// TIA Portal V19 export
DATA_BLOCK "ALARM DB"   // DB20
{ S7_Optimized_Access := 'FALSE' }
   VAR
      "EMERGENCY STOP" : Bool;
      "AIR FAIL" : Bool;
      "MGF FEED PUMP P-101 A MCB TRIP" : Bool;
      "MGF FEED PUMP P-101 B MCB TRIP" : Bool;
      "MGF BACK WASH  P-102 A MCB TRIP" : Bool;
      "MGF BACK WASH P-102 B MCB TRIP" : Bool;
      "UF FEED PUMP P-103 A MCB TRIP" : Bool;
      "UF FEED PUMP P-103 B MCB TRIP" : Bool;
      "UF BLOWER AB-201 A MCB TRIP" : Bool;
      "UF BLOWER AB-201 B MCB TRIP" : Bool;
      "DM FEED PUMP P-502 A MPCB TRIP" : Bool;
      "DM FEED PUMP P-502 B MPCB TRIP" : Bool;
      "DM FEED PUMP P-502 C MPCB TRIP" : Bool;
      "CIP P-601" : Bool;
      "BACK WASH RECOVERY P-801 A MPCB TRIP" : Bool;
      "BACK WASH RECOVERY P-801 B MPCB TRIP" : Bool;
      "UF BACKWASH P-201A TRIP" : Bool;
      "UF BACKWASH P-201B TRIP" : Bool;
      "MGF FEED PUMP P-101 A MCB_FEEDBACK FAIL" : Bool;
      "MGF FEED PUMP P-101 B MCB_FEEDBACK FAIL" : Bool;
      "MGF BACK WASH  P-102 A MCB_FEEDBACK FAIL" : Bool;
      "MGF BACK WASH P-102 B MCB_FEEDBACK FAIL" : Bool;
      "UF FEED PUMP P-103 A MCB_FEEDBACK FAIL" : Bool;
      "UF FEED PUMP P-103 B MCB_FEEDBACK FAIL" : Bool;
      "UF BLOWER AB-201 A MCB_FEEDBACK FAIL" : Bool;
      "UF BLOWER AB-201 B MCB_FEEDBACK FAIL" : Bool;
      "DM FEED PUMP P-502 A MPCB_FEEDBACK FAIL" : Bool;
      "DM FEED PUMP P-502 B MPCB_FEEDBACK FAIL" : Bool;
      "DM FEED PUMP P-502 C MPCB_FEEDBACK FAIL" : Bool;
      "CIP P-601_FEEDBACK FAIL" : Bool;
      "BACK WASH RECOVERY P-801 A MPCB_FEEDBACK FAIL" : Bool;
      "BACK WASH RECOVERY P-801 B MPCB_FEEDBACK FAIL" : Bool;
      "UF BACKWASH P-201A_FEEDBACK FAIL" : Bool;
      "UF BACKWASH P-201B_FEEDBACK FAIL" : Bool;
      "MGF INLET VALVE ABFV-101 OPEN COMMOND FAIL" : Bool;
      "MGF INLET VALVE ABFV-101 CLOSE COMMOND FAIL" : Bool;
      "MGF BACKWASH OUTLET VALVE ABFV-102 OPEN COMMOND FAIL" : Bool;
      "MGF BACKWASH OUTLET VALVE ABFV-102 CLOSE COMMOND FAIL" : Bool;
      "MGF BACKWASH INLET VALVE ABFV-103 OPEN COMMOND FAIL" : Bool;
      "MGF BACKWASH INLET VALVE ABFV-103 CLOSE COMMOND FAIL" : Bool;
      "MGF OUTLET VALVE ABFV-104 OPEN COMMOND FAIL" : Bool;
      "MGF OUTLET VALVE ABFV-104 CLOSE COMMOND FAIL" : Bool;
      "MGF RINSE OUTLET VALVE ABFV-105 OPEN COMMOND FAIL" : Bool;
      "MGF RINSE OUTLET VALVE ABFV-105 CLOSE COMMOND FAIL" : Bool;
      "UF AIR SCOURING VALVE ABV-201 OPEN COMMOND FAIL" : Bool;
      "UF AIR SCOURING VALVE ABV-201 CLOSE COMMOND FAIL" : Bool;
      "UF INLET VALVE ABFV-201 OPEN COMMOND FAIL" : Bool;
      "UF INLET VALVE ABFV-201 CLOSE COMMOND FAIL" : Bool;
      "UF BOTTOM DAIN VALVE ABFV-202 OPEN COMMOND FAIL" : Bool;
      "UF BOTTOM DAIN VALVE ABFV-202 CLOSE COMMOND FAIL" : Bool;
      "UF TOP DAIN VALVE ABFV-203 OPEN COMMOND FAIL" : Bool;
      "UF TOP DAIN VALVE ABFV-203 CLOSE COMMOND FAIL" : Bool;
      "UF BACKWASH INLET VALVE ABFV-204 OPEN COMMOND FAIL" : Bool;
      "UF BACKWASH INLET VALVE ABFV-204 CLOSE COMMOND FAIL" : Bool;
      "UF PRODUCT OUT VALVE ABFV-205 OPEN COMMOND FAIL" : Bool;
      "UF PRODUCT OUT VALVE ABFV-205 CLOSE COMMOND FAIL" : Bool;
      "UF BACKWASH RECOVERY LINE VALVE ABFV-206 OPEN COMMOND FAIL" : Bool;
      "UF BACKWASH RECOVERY LINE VALVE ABFV-206 CLOSE COMMOND FAIL" : Bool;
      "UF BACKWASH DRAIN LINE VALVE ABFV-207 OPEN COMMOND FAIL" : Bool;
      "UF BACKWASH DRAIN LINE VALVE ABFV-207 CLOSE COMMOND FAIL" : Bool;
      "UF BACKWASH BYPASS VALVE ABFV-208 OPEN COMMOND FAIL" : Bool;
      "UF BACKWASH BYPASS VALVE ABFV-208 CLOSE COMMOND FAIL" : Bool;
      "RAW WATER COLLECTION TANK LEVEL ( LT-101)- LOW LOW" : Bool;
      "RAW WATER COLLECTION TANK LEVEL ( LT-101)- HIGH HIGH" : Bool;
      "FILTER WATER STORAGE TANK  LEVEL ( LT-102)- LOW LOW" : Bool;
      "FILTER WATER STORAGE TANK LEVEL ( LT-102)- HIGH HIGH" : Bool;
      "RO-01 FEED TANK LEVEL ( LT-201)- LOW LOW" : Bool;
      "RO-01 FEED TANK LEVEL ( LT-201)- HIGH HIGH" : Bool;
      "BACKWASH WASTE WATER COLLECTION TANK  LEVEL ( LT-801)- LOW LOW" : Bool;
      "BACKWASH WASTE WATER COLLECTION TANK LEVEL ( LT-801)- HIGH HIGH" : Bool;
      "PS-201 HIGH" : Bool;
      "DPT-101 HIGH" : Bool;
      "DPT-201 HIGH" : Bool;
      "NRMB OUTLET PRESSURE PT-601 HIGH" : Bool;
      "NRMB PRODUCT OUT pHIT-601 HIGH" : Bool;
      "NRMB PRODUCT OUT pHIT-601 LOW" : Bool;
      "NRMB PRODUCT OUT RIT-601 HIGH" : Bool;
      "RIT-601 HIGH_SET VALIDATION TIME OVER_(SYSTEM STOP)" : Bool;
      "UV-601 INTENSITY LOW" : Bool;
   END_VAR
BEGIN
END_DATA_BLOCK
